FUNCTION_BLOCK Codes_StopReason
VAR_INPUT
	EN: BOOL;
	StopButton_Num : INT;       
END_VAR
VAR_OUTPUT
	ENO: BOOL;
	Code_Valid: BOOL;
	Code_StopReason : STRING;  
	
	
END_VAR
VAR
	
END_VAR

IF NOT EN THEN
    ENO := FALSE;
    Code_StopReason := '';
    Code_Valid := FALSE;
    RETURN;
END_IF

ENO := TRUE;

CASE StopButton_Num OF
    10: Code_StopReason := 'MNT_C01';
    20: Code_StopReason := 'MNT_G01';
    30: Code_StopReason := 'MSP_C01';
    40: Code_StopReason := 'MSP_P01';
    50: Code_StopReason := 'QLT_Q01';
    60: Code_StopReason := 'TEC_E0M';
	70: Code_StopReason := 'MSP_F01';
ELSE
    Code_StopReason := '';
END_CASE;

Code_Valid := (Code_StopReason <> '');

END_FUNCTION_BLOCK

(* stored: Version 1.1.0.1, ProductVersion 3.1.4024.15
   POU Codes_StopReason: Id {b668e012-512e-40ed-91d5-bae83592be95}, SpecialFunc None *)
